(* CODESYS project rsCommTcpRt.library
   Company: ESO
   Description: This library provides generic drivers for Tcp Real-time communication.
      It also provides Local Control Device drivers for Tcp Real-time communication with Lakeshore 224 and 336.
      Depends on rsCommCommon.library
   Version: 0.2.0.3
   Placeholder: ESO LDC Comm Tcp RT Library
   Author: Dan Popovic
   Title: ESO LDC Comm Tcp RT Library

Project tree, tasks and I/O mapping:
  libraries: ESO LDC Comm Common Library, 0.2.0.3 (ESO); Tc2_Standard, * (Beckhoff Automation GmbH); Tc2_System, * (Beckhoff Automation GmbH); Tc2_Utilities, * (Beckhoff Automation GmbH); Tc3_Module, * (Beckhoff Automation GmbH); VisuDialogs, * (System); VisuSymbols, * (System)
  config/
    Lakeshore_RT_Ethernet_Adapter_InterfacePointer.jpg
    Lakeshore_RT_Ethernet_Adapter_Params.jpg
    Lakeshore_RT_Instance_OID_SymbolInitialization.png
  00000000-0000-0000-0000-000000000000|config\Lakeshore_RT_Ethernet_Adapter_InterfacePointer.jpg
  00000000-0000-0000-0000-000000000000|config\Lakeshore_RT_Ethernet_Adapter_Params.jpg
  00000000-0000-0000-0000-000000000000|config\Lakeshore_RT_Instance_OID_SymbolInitialization.png
  Data types/
    Enumerated/
      Comm/
        data type E_TCP_RT_CLIENT_STATUS
    Structures/
      Comm/
        data type T_TCP_RT_CLIENT_CFG
        data type T_TCP_RT_CLIENT_CTRL
        data type T_TCP_RT_CLIENT_INFO
        data type T_TCP_RT_CLIENT_STAT
        data type U_IpAdr
  Global Variables/
  lib/
  POUs/
    Comm/
      function block FB_TCP_RT_CLIENT [ST]: FB_exit, FB_init, FB_reinit, ReceiveData, ReceiveEvent, TcAddRef, TcQueryInterface, TcRelease
    Devices/
      function block FB_LAKESHORE_TCP_RT [ST]: ActivityInitializing, ActivityMonitoring, ActivityMonitoringUser, M_Configure, M_GetCouplerState, M_ReadFromReply, M_ReadSensors, M_UpdateStatus
    program MAIN [ST]
  Version/
    global variables Global_Version
  Visualizations/
    Templates/
      visualisation GUI_TEMPLATE_LAKESHORE_TCP_RT_224
      visualisation GUI_TEMPLATE_LAKESHORE_TCP_RT_336
    visualisation GUI_LAKESHORE_TCP_RT_224
    visualisation GUI_LAKESHORE_TCP_RT_336
  text list GlobalTextList
*)

// Data types/Enumerated/Comm/E_TCP_RT_CLIENT_STATUS
{attribute 'qualified_only'}
{attribute 'strict'}
TYPE E_TCP_RT_CLIENT_STATUS :
(
	NOT_INIT	:= -1,
	IDLE		:= 0,
	BUSY		:= 1,
	ERROR		:= 2
);
END_TYPE

// Data types/Structures/Comm/T_TCP_RT_CLIENT_CFG
TYPE T_TCP_RT_CLIENT_CFG :
STRUCT
	sTcpServerAdr:	STRING(16)	:= '62.159.14.51';	// Beckhoff Test-Website
    nTcpPort:    	UINT := 80;						// Beckhoff Test-Website
	

	// Parameters hidden from OPC UA access
	{attribute 'OPC.UA.DA' := '0'}
	tcpServerAdr:	U_IpAdr; 
END_STRUCT
END_TYPE

// Data types/Structures/Comm/T_TCP_RT_CLIENT_CTRL
TYPE T_TCP_RT_CLIENT_CTRL :
STRUCT
	bExecute: 	BOOL 	:= FALSE;
	sCmd:		STRING;
END_STRUCT
END_TYPE

// Data types/Structures/Comm/T_TCP_RT_CLIENT_INFO
TYPE T_TCP_RT_CLIENT_INFO :
STRUCT
(*
	Driver Information

	Change LOG:
	0.1.0.0		- First version.
*)

	sDate:			STRING(32)	:= '2018-10-09';
	sDescription:	STRING(80) 	:= 'TCP Client RT';
	sName:			STRING(64)	:= 'FB_TCP_CLIENT';
	sPlatform:		STRING(32)	:= 'CoDeSys';
	sSynopsis:		STRING(64)	:= 'TCP Client RT';
	nVersionMajor:	DINT		:= 0;
	nVersionMinor:	DINT		:= 1;

END_STRUCT
END_TYPE

// Data types/Structures/Comm/T_TCP_RT_CLIENT_STAT
TYPE T_TCP_RT_CLIENT_STAT :
STRUCT
	bInitialised:		BOOL	:= FALSE;		(* Flag if device is initialised *)


	nLastCommand:		DINT 	:= 0;
	nErrorCode:			DINT 	:= 0;
	nStatus: 			DINT	:= E_TCP_RT_CLIENT_STATUS.NOT_INIT;	// IDLE, BUSY, ERROR
	nCounter:			UDINT	:= 0;	// Alive counter

	sErrorText: 		STRING 	:= 'OK';
	sStatus:			STRING	:= '';	// Status description

	sLibVersion:		STRING	:= 'UNKNOWN';					(* Library version, e.g. '1.2.0.0' *)
	sSvnRevision:		STRING	:= '$$Revision: 311362 $$';		(* SVN Revision *)
	sRevision:			STRING	:= '';							(* SVN Revision without $ signs *)

	//Sample information about communication
    nReceivedPakets:	UINT;

	nSocketId:			UDINT; 
	nSentData:			UDINT; 

	bConnected:			BOOL	:= FALSE;
	nConnections: 		UDINT; 
	lastTcpEvent: 		TCPIP_EVENT;
	nReplyLength: 		UDINT; 
	sReply: 			STRING(255); 
	hrSend: 			HRESULT; //last SendData result

END_STRUCT
END_TYPE

// Data types/Structures/Comm/U_IpAdr
TYPE U_IpAdr :
UNION
	ipadrInternal : UDINT;
	ipadr : ARRAY[0..3] OF BYTE;
END_UNION
END_TYPE

// Version/Global_Version
{attribute 'TcGenerated'}
{attribute 'no-analysis'}
{attribute 'linkalways'}
// This function has been automatically generated from the project information.
VAR_GLOBAL CONSTANT
	{attribute 'const_non_replaced'}
	stLibVersion_ESO_LDC_Comm_Tcp_RT_Library : ST_LibVersion := (iMajor := 0, iMinor := 2, iBuild := 0, iRevision := 3, nFlags := 0, sVersion := '0.2.0.3');
END_VAR

// POUs/Comm/FB_TCP_RT_CLIENT
{attribute 'c++_compatible'}
FUNCTION_BLOCK FB_TCP_RT_CLIENT IMPLEMENTS ITcIoTcpProtocolRecv
VAR_INPUT
	{attribute 'OPC.UA.DA' := '0'}
	in_sDeviceTcpIpAdr:	STRING(16);	// Device IP address, e.g. '192.168.0.80'
	{attribute 'OPC.UA.DA' := '0'}
    in_nDeviceTcpPort:  UINT;		// Device Tcp port
END_VAR
VAR_OUTPUT
END_VAR
VAR
	{attribute 'OPC.UA.DA' := '1'}
	cfg:		T_TCP_RT_CLIENT_CFG;				// Config parameters
	{attribute 'OPC.UA.DA' := '1'}
	ctrl:		T_TCP_RT_CLIENT_CTRL;				// Control parameters
	{attribute 'OPC.UA.DA' := '1'}
	{attribute 'OPC.UA.DA.Access' := '1'}
	info:		T_TCP_RT_CLIENT_INFO; 				// Info parameters - ReadOnly
	{attribute 'OPC.UA.DA' := '1'}
	{attribute 'OPC.UA.DA.Access' := '1'}
	stat:		T_TCP_RT_CLIENT_STAT;				// Status parameters - ReadOnly


	// The following attribute has to be linked to corresponding Value 
	// of RT-Ethernet Adapter in Instance/'Symbol Initialization' tab
	{attribute 'TcInitSymbol'}
    oid: OTCID;	// Link to Value of RT-Ethernet Adapter in Instance/'Symbol Initialization' tab
	
    ipTcp:       ITcIoTcpProtocol;
	
	// Local variables
    ids: 	T_IPv4AddrArr;
	hrInit:	HRESULT; 
	
	// In case of error, try to allocate socket on every 100-th cycle.
	nSocketCounter:	UINT	:= 0;
	nSocketCounterLimit:	UINT	:= 100;
	

END_VAR

// TODO: Complete configuration
IF NOT stat.bInitialised THEN
	// Copy input parameters to config
	cfg.sTcpServerAdr	:= in_sDeviceTcpIpAdr;
	cfg.nTcpPort		:= in_nDeviceTcpPort;
	
	//generate Server IP adress
	ids := F_ScanIPv4AddrIds( in_sDeviceTcpIpAdr ); 
	cfg.tcpServerAdr.ipadr[3] := ids[0]; 
	cfg.tcpServerAdr.ipadr[2] := ids[1]; 
	cfg.tcpServerAdr.ipadr[1] := ids[2];
	cfg.tcpServerAdr.ipadr[0] := ids[3];
	
	// Get the version number 
	stat.sLibVersion	:= Global_Version.stLibVersion_ESO_LDC_Comm_Tcp_RT_Library.sVersion;
	stat.sRevision		:= MID(stat.sSvnRevision, LEN(stat.sSvnRevision)-2, 2);

	stat.bInitialised	:= TRUE;
	RETURN;
END_IF

IF(ipTcp <> 0) THEN 
	ipTcp.CheckReceived(); 
	IF (stat.nSocketId = 0) THEN 
		stat.bConnected	:= FALSE;
		nSocketCounter	:= nSocketCounter + 1;
		IF nSocketCounter > nSocketCounterLimit THEN
			nSocketCounter	:= 0;
			IF(ipTcp.AllocSocket(THIS^, stat.nSocketId) = 0) THEN //! THIS^ might get invalid due to online change! "Reallocate" by nSocketId <>0
				stat.nConnections := stat.nConnections+1;
				IF(ipTcp.Connect(stat.nSocketId, cfg.tcpServerAdr.ipadrInternal, cfg.nTcpPort) <> 0) THEN
					ipTcp.FreeSocket(stat.nSocketId); 
					stat.nSocketId := 0; 
				END_IF
			END_IF
		END_IF
	ELSE
		IF (ipTcp.IsConnected(stat.nSocketId) = S_OK) THEN 
			stat.bConnected	:= TRUE;
			IF ctrl.bExecute THEN
				ctrl.bExecute := FALSE;
				stat.hrSend := ipTcp.SendData(stat.nSocketId, INT_TO_UDINT(LEN(ctrl.sCmd)), ADR(ctrl.sCmd), stat.nSentData); 
			END_IF
		ELSE
			IF stat.bConnected THEN
				// We were connected but not any more.
				// Free the socket.
				ipTcp.FreeSocket(stat.nSocketId); 
				stat.nSocketId := 0; 
			END_IF
			stat.bConnected	:= FALSE;
		END_IF
	END_IF
END_IF

METHOD FB_exit : BOOL
VAR_INPUT
	bInCopyCode : BOOL; // if TRUE, the exit method is called for exiting an instance that is copied afterwards (online change).
END_VAR
IF NOT bInCopyCode THEN // no online change
	IF ipTcp <> 0 THEN 
		ipTcp.FreeSocket(stat.nSocketId); // Shutdown
		FW_SafeRelease(ADR(ipTcp));
		FB_exit := TRUE; 
	END_IF
END_IF
END_METHOD

METHOD FB_init : BOOL
VAR_INPUT
	bInitRetains: 	BOOL; // if TRUE, the retain variables are initialized (warm start / cold start)
	bInCopyCode: 	BOOL;  // if TRUE, the instance afterwards gets moved into the copy code (online change)
END_VAR
VAR
	ipSrv:	ITComObjectServer;
	
END_VAR
IF NOT bInCopyCode THEN // no online change
	IF ipTcp = 0 THEN
		hrInit := FW_ObjMgr_GetObjectInstance(	oid:=oid, 
												iid:=TC_GLOBAL_IID_LIST.IID_ITcIoTcpProtocol, 
												pipUnk:=ADR(ipTcp) );
		IF SUCCEEDED(hrInit) THEN
			FB_init := TRUE;
		ELSE 
			FW_SafeRelease(ADR(ipTcp));
		END_IF 
	END_IF
END_IF
END_METHOD

METHOD FB_reinit : BOOL
VAR_INPUT
END_VAR
IF (ipTcp <> 0 AND stat.nSocketId <> 0) THEN //reregister THIS^ for online changes  
	ipTcp.AllocSocket(THIS^, stat.nSocketId);
	FB_reinit := TRUE; 
END_IF
END_METHOD

{attribute 'object_name' := 'ReceiveData'}
{attribute 'c++_compatible'}
{attribute 'signature_flag' := '33554688'}
{attribute 'pack_mode' := '4'}
{attribute 'show'}
{attribute 'minimal_input_size' := '4'}
{attribute 'checksuperglobal'}
METHOD ReceiveData : HRESULT
VAR_INPUT
	socketId	: UDINT;
	nData	: UDINT;
	pData	: PVOID;
END_VAR
stat.nReceivedPakets	:= stat.nReceivedPakets+1;
stat.nReplyLength 		:= nData; //nonstripped

MEMCPY( ADR(stat.sReply), pData, MIN(nData, SIZEOF(stat.sReply)-1) );	//stripped to max length of string
memset(ADR(stat.sReply)+MIN(nData, SIZEOF(stat.sReply)-1)+1, 0, 1);		//add a 00 Byte at end of message
END_METHOD

{attribute 'object_name' := 'ReceiveEvent'}
{attribute 'c++_compatible'}
{attribute 'signature_flag' := '33554688'}
{attribute 'pack_mode' := '4'}
{attribute 'show'}
{attribute 'minimal_input_size' := '4'}
{attribute 'checksuperglobal'}
METHOD ReceiveEvent : HRESULT
VAR_INPUT
	socketId	: UDINT;
	tcpEvent	: TCPIP_EVENT;
END_VAR
stat.lastTcpEvent := tcpEvent;

CASE tcpEvent OF
	TCPIP_EVENT.TCPIP_EVENT_ERROR:
		stat.nStatus	:= E_TCP_RT_CLIENT_STATUS.ERROR;
		stat.sStatus	:= 'ERROR';
		ipTcp.FreeSocket(socketId);
		stat.nSocketId := 0; 
	TCPIP_EVENT.TCPIP_EVENT_RESET:
		stat.nStatus	:= E_TCP_RT_CLIENT_STATUS.BUSY;
		ipTcp.FreeSocket(socketId);
		stat.nSocketId := 0; 
	TCPIP_EVENT.TCPIP_EVENT_TIMEOUT:
		stat.nStatus	:= E_TCP_RT_CLIENT_STATUS.ERROR;
		stat.sStatus	:= 'TIMEOUT';
		ipTcp.FreeSocket(socketId);
		stat.nSocketId := 0; 
	TCPIP_EVENT.TCPIP_EVENT_CONN_CLOSED:
		ipTcp.FreeSocket(socketId);
		stat.nSocketId := 0; 
	TCPIP_EVENT.TCPIP_EVENT_CONN_INCOMING:
		stat.nStatus	:= E_TCP_RT_CLIENT_STATUS.BUSY;
	TCPIP_EVENT.TCPIP_EVENT_KEEP_ALIVE:
		stat.nStatus	:= E_TCP_RT_CLIENT_STATUS.BUSY;
	TCPIP_EVENT.TCPIP_EVENT_CONN_IDLE:
(*
		// Recovery
		IF ctrl.bExecute THEN
			ctrl.bExecute	:= FALSE;
			THIS^.ReceiveEvent(socketId,TCPIP_EVENT.TCPIP_EVENT_RESET);
		ELSE
			stat.nStatus	:= E_TCP_RT_CLIENT_STATUS.IDLE;
		END_IF
*)
	TCPIP_EVENT.TCPIP_EVENT_DATA_SENT:
		stat.sStatus	:= CONCAT(ctrl.sCmd, ' Sent');
	TCPIP_EVENT.TCPIP_EVENT_DATA_RECEIVED:
		stat.nStatus	:= E_TCP_RT_CLIENT_STATUS.IDLE;
		stat.sStatus	:= 'Data Received';
	(*
		IF nCmd = 1 THEN
			ctrl.sMessage	:= 'PID? 1$N';
			nCmd	:= 2;
		ELSIF nCmd = 2 THEN
			ctrl.sMessage	:= 'PID? 2$N';
			nCmd	:= 1;
		END_IF
		ctrl.bSend	:= TRUE;
		*)
//		THIS^.ReceiveEvent(socketId,TCPIP_EVENT.TCPIP_EVENT_CONN_IDLE);
	TCPIP_EVENT.TCPIP_EVENT_LINKCONNECT:
	// WARNING: Nothing to do?
	TCPIP_EVENT.TCPIP_EVENT_LINKDISCONNECT:
		ipTcp.FreeSocket(socketId);
		stat.nSocketId := 0; 
END_CASE; 
ReceiveEvent := S_OK;
END_METHOD

{attribute 'object_name' := 'TcAddRef'}
{attribute 'c++_compatible'}
{attribute 'signature_flag' := '33554688'}
{attribute 'pack_mode' := '4'}
{attribute 'show'}
{attribute 'minimal_input_size' := '4'}
{attribute 'checksuperglobal'}
METHOD TcAddRef : UDINT
END_METHOD

{attribute 'object_name' := 'TcQueryInterface'}
{attribute 'c++_compatible'}
{attribute 'signature_flag' := '33554688'}
{attribute 'pack_mode' := '4'}
{attribute 'show'}
{attribute 'minimal_input_size' := '4'}
{attribute 'checksuperglobal'}
METHOD TcQueryInterface : HRESULT
VAR_INPUT
	iid	: REFERENCE TO IID;
	pipItf	: POINTER TO PVOID;
END_VAR
VAR
	ipTcpRecv : ITcIoTcpProtocolRecv;
	ipUnknown : ITcUnknown;	
END_VAR
IF GuidsEqual(ADR(iid), ADR(TC_GLOBAL_IID_LIST.IID_ITcIoTcpProtocolRecv)) THEN
	ipTcpRecv := THIS^; // cast to interface pointer
	pipItf^ := ITCUNKNOWN_TO_PVOID(ipTcpRecv);
	TcAddRef();
	TcQueryInterface := S_OK;
ELSIF GuidsEqual(ADR(iid), ADR(TC_GLOBAL_IID_LIST.IID_ITcUnknown)) THEN
	ipUnknown := THIS^; // cast to interface pointer
	pipItf^ := ITCUNKNOWN_TO_PVOID(ipUnknown);
	TcAddRef();
	TcQueryInterface := S_OK;
ELSE
	TcQueryInterface := E_HRESULTAdsErr.NOINTERFACE ; //Call super if this fb extends some other
END_IF
END_METHOD

{attribute 'object_name' := 'TcRelease'}
{attribute 'c++_compatible'}
{attribute 'signature_flag' := '33554688'}
{attribute 'pack_mode' := '4'}
{attribute 'show'}
{attribute 'minimal_input_size' := '4'}
{attribute 'checksuperglobal'}
METHOD TcRelease : UDINT
END_METHOD

END_FUNCTION_BLOCK

// POUs/Devices/FB_LAKESHORE_TCP_RT
FUNCTION_BLOCK FB_LAKESHORE_TCP_RT EXTENDS FB_LAKESHORE_BASE
VAR_INPUT
	{attribute 'OPC.UA.DA' := '0'}
	in_sDeviceTcpIpAdr:	STRING(16);		// Lakeshore IP address, e.g. '192.168.0.80'
	{attribute 'OPC.UA.DA' := '0'}
    in_nDeviceTcpPort:  UINT := 7777;	// Lakeshore Tcp port, default 7777
END_VAR
VAR_OUTPUT
END_VAR
VAR CONSTANT
	// Monitoring states
	{attribute 'OPC.UA.DA' := '0'}
	C_STATE_SEND_CMD:			INT	:= 0;
	{attribute 'OPC.UA.DA' := '0'}
	C_STATE_DELAY_AFTER_SEND:	INT	:= 10;
	{attribute 'OPC.UA.DA' := '0'}
	C_STATE_WAIT_DATA_RECEIVED:	INT	:= 20;
	{attribute 'OPC.UA.DA' := '0'}
	C_STATE_WAIT:				INT	:= 30;
END_VAR
VAR

	{attribute 'OPC.UA.DA' := '0'}
	comm:		FB_TCP_RT_CLIENT;			// Instance of generic comm FB. OPC UA Disabled!!!

END_VAR


(* Execute comm instance *)
comm(	in_sDeviceTcpIpAdr:=in_sDeviceTcpIpAdr,
		in_nDeviceTcpPort:=in_nDeviceTcpPort);


// Execute the base class object FB_RS_BASE
SUPER^();

METHOD ActivityInitializing
VAR_INPUT
	bExecute:	BOOL;
END_VAR
VAR_INST
	{attribute 'OPC.UA.DA' := '0'}
    nMethodState:	INT := 0;	// State Machine current state
END_VAR
SetAction('ActivityInitializing');


IF NOT bExecute THEN
	nMethodState	:= 0;	// Reset the state machine
	cmdCounter		:= 1;	// Init will start from the first init command
	RETURN;
END_IF

// Handle State Machine
CASE nMethodState OF
	0:	// Set communication parameters and Model configuration
		(* Set comm suffixes for commands and replies *)
		// TODO: Suffix
//		ptrCommCfg^.sCmdSuffix		:= sCmdSuffix;
//		ptrCommCfg^.sReplySuffix	:= sReplySuffix;
		// Set Model and monitoring period (input parameters)
		cfg.nModel			:= in_nModel;
		cfg.bAutoMonitor	:= in_bAutoMonitor;
		cfg.tDelay_Periodic	:= DINT_TO_TIME(in_nPeriod);
		
		(* Pointers to INIT and READ commands set in M_Configure() depending on the model *)

		(* Set initial state and status *)
		stat.bInitialised	:= FALSE;
		stat.sReply			:= '';
		SetStatus(E_SM_ERROR.OK, 'BUSY');
		
		// DPO NEW START
		// Wait for connected
		fbTimer (IN := FALSE); (* Reset timer *)
		fbTimer (IN := TRUE, PT := T#10S); (* TODO: 80 sec timeout for reply *)
		nMethodState := 5;				// Go to next state, i.e. INIT_COMM
		RETURN;
		// DPO NEW END

		nMethodState := 10;				// Go to next state, i.e. INIT_COMM
		
		
	5:
		fbTimer (IN := TRUE);
		IF fbTimer.Q THEN
			// Timer expired after 5 sec. This is an error.
			fbTimer (IN := FALSE);
			SetStatus(E_LAKESHORE_ERROR.TIMEOUT, 'ERROR: Communication timeout');	
			bCommProblem	:= TRUE;
			nEvent := E_SM_EVENT.ERRINIT;
			RETURN;
		ELSIF comm.stat.bConnected THEN
			fbTimer (IN := FALSE);
			nMethodState := 10;				// Go to next state, i.e. INIT_COMM
		END_IF

	10:	// Initialize COMM port
		(* Reset the serial port *)
//		ptrCommCtrl^.nCommand	:= E_RS_COMM_CMD.INIT;
//		ptrCommCtrl^.bExecute	:= TRUE;

		(* Start the timer by going false/true *)
		fbTimer (IN := FALSE); (* Reset timer *)
		fbTimer (IN := TRUE, PT := T#20S); (* TODO: 80 sec timeout for reply *)

//		nMethodState 	:= 15;	// On next cycle wait until the comm port is reset, i.e. idle
		nMethodState 	:= 20;	// On next cycle wait until the comm port is reset, i.e. idle
		
	15:	// Wait for completion of command.
		// If command has no reply, wait for comm.stat.lastTcpEvent = TCPIP_EVENT.TCPIP_EVENT_DATA_SENT.
		// If it has, wait for               comm.stat.lastTcpEvent = TCPIP_EVENT.TCPIP_EVENT_DATA_RECEIVED.
		fbTimer (IN := TRUE);
		IF ((cfg.cmdList_Init[cmdCounter].nReplies = 0) AND 
			(comm.stat.lastTcpEvent = TCPIP_EVENT.TCPIP_EVENT_DATA_SENT OR 
			 comm.stat.lastTcpEvent = TCPIP_EVENT.TCPIP_EVENT_CONN_IDLE)) OR 
			((cfg.cmdList_Init[cmdCounter].nReplies > 0) AND 
			(comm.stat.lastTcpEvent = TCPIP_EVENT.TCPIP_EVENT_DATA_RECEIVED))THEN
			// Communication is IDLE 
			fbTimer (IN := FALSE);	// disable timer 
			stat.sReply		:= ptrCommStat^.sReply;	// Save the reply
			cmdCounter		:= cmdCounter + 1;	// Increment init command index
			fbTimer (IN := FALSE);	// disable timer 
			fbTimer (IN := TRUE, PT := cfg.tDelay_Init); // Wait INIT delay
			bCommProblem	:= FALSE;
			nMethodState 	:= 18;	// Execute next device INIT command
		ELSIF comm.stat.nStatus = E_RS_COMM_STATUS.ERROR THEN
			fbTimer (IN := FALSE);
			SetStatus(E_LAKESHORE_ERROR.COMM, 'ERROR: Communication error');	
			bCommProblem	:= TRUE;
			nEvent := E_SM_EVENT.ERRINIT;
			RETURN;
		ELSIF fbTimer.Q THEN
			// Timer expired after 5 sec. This is an error.
			fbTimer (IN := FALSE);
			SetStatus(E_LAKESHORE_ERROR.TIMEOUT, 'ERROR: Communication timeout');	
			bCommProblem	:= TRUE;
			nEvent := E_SM_EVENT.ERRINIT;
			RETURN;
		END_IF

	
	
	18:	// Wait INIT Delay
		fbTimer (IN := TRUE);
		IF fbTimer.Q THEN
			// Timer expired after 5 sec. This is an error.
			fbTimer (IN := FALSE);
			nMethodState 	:= 20;	// Execute next device INIT command
			RETURN;
		END_IF

	
	
	20:	// INIT DEV
		IF cfg.cmdList_Init[cmdCounter].cmd = '' THEN
			// Device INIT is done. Go to IDLE 
			stat.bInitialised 	:= TRUE;
			cmdCounter			:= 1;
			SetStatus(E_SM_ERROR.OK, 'IDLE');
			nEvent 		:= E_SM_EVENT.INITDONE;
			RETURN;
		END_IF
		
		(* Send INIT command with index cmdCounter *)
//		ptrCommCtrl^.nCommand		:= E_RS_COMM_CMD.SEND;
		ptrCommCtrl^.sCmd			:= CONCAT(cfg.cmdList_Init[cmdCounter].cmd,in_sCmdSuffix);
//		ptrCommCtrl^.nNumReplies	:= ptrInitCmds^ [cmdCounter].nReplies;
//		ptrCommCtrl^.bHasReply		:= ptrInitCmds^ [cmdCounter].nReplies > 0;
		ptrCommCtrl^.bExecute		:= TRUE;
	
		(* Start the timer by going false/true *)
		fbTimer (IN := FALSE); (* Reset timer *)
		fbTimer (IN := TRUE, PT := T#5S); (* 5 sec timeout for reply *)

		// On next cycle wait until the comm port is idle
		nMethodState 	:= 15;	// On next cycle wait until the comm port is idle
	
END_CASE
END_METHOD

METHOD ActivityMonitoring
VAR_INPUT
	bExecute:	BOOL;
END_VAR
VAR_INST
	{attribute 'OPC.UA.DA' := '0'}
    nMethodState:	INT := C_STATE_SEND_CMD;	// State Machine current state
	{attribute 'OPC.UA.DA' := '0'}
	nRetries:		INT := 0;	// Number of retries in case of communication problems
	{attribute 'OPC.UA.DA' := '0'}
	tDelay:			TIME	:= T#50MS;	// Min delay to wait after a command
END_VAR
IF NOT cfg.bAutoMonitor AND stat.nSubstate = E_RS_BASE_SUBSTATE.NOTOP_READY THEN
	SetAction('No Monitoring'); 
	SetStatus(E_SM_ERROR.OK, 'IDLE');
	nMethodState	:= C_STATE_SEND_CMD;	// Reset the state machine
	cmdCounter		:= 1;	// Reading will start from the first command in the array
	RETURN;
END_IF

IF NOT bExecute THEN
	SetAction('ActivityMonitoring'); 
//	SetStatus(E_SM_ERROR.OK, 'BUSY');
	nMethodState	:= C_STATE_SEND_CMD;	// Reset the state machine
	cmdCounter		:= 1;	// Reading will start from the first command in the array
	RETURN;
END_IF

// Handle State Machine
CASE nMethodState OF
	/////////////////
	C_STATE_SEND_CMD:	// Execute a command from the command array
	/////////////////
		IF cfg.cmdList_Read[cmdCounter].cmd = '' OR cmdCounter > 16 THEN
			// We arrived to the end of the array of pre-defined commands
			// Check if we have to exit Monitoring
			IF nReadType = E_RS_BASE_READ_TYPE.SINGLE	THEN
				// If it's a single read, exit here.
				SetStatus(E_SM_ERROR.OK, 'IDLE');
				nInternalEvent := E_SM_EVENT.READDONE;
				RETURN;
			END_IF

			// Periodic READ is done. Wait tDelay_Periodic before re-starting the READ.
			cmdCounter	:= 1;
			SetStatus(E_SM_ERROR.OK, 'IDLE');
			
			(* Start the timer by going false/true *)
			fbTimer (IN := FALSE); (* Reset timer *)
			fbTimer (IN := TRUE, PT := cfg.tDelay_Periodic);
			nMethodState := C_STATE_WAIT;				// Goto Wait for tDelay_Periodic
			RETURN;
		ELSIF NOT comm.stat.bConnected THEN
			SetStatus(E_LAKESHORE_ERROR.COMM, 'Send Failed.');	
			// Not connected yet. Don't do anything
			(* Start the timer by going false/true *)
			fbTimer (IN := FALSE); (* Reset timer *)
			fbTimer (IN := TRUE, PT := T#3S);
			nMethodState := C_STATE_WAIT;				// Goto Wait for tDelay_Periodic
			nEvent := E_SM_EVENT.ERRCOMM;
			RETURN;
		ELSE
			(* Send command with index cmdCounter *)
			ptrCommCtrl^.sCmd		:= CONCAT(cfg.cmdList_Read[cmdCounter].cmd,in_sCmdSuffix);
			ptrCommCtrl^.bExecute	:= TRUE;
			
			(* Start the timer by going false/true *)
			fbTimer (IN := FALSE); (* Reset timer *)
			fbTimer (IN := TRUE, PT := T#3MS); // 3 msec timeout before waiting for reply 
	
			nMethodState := C_STATE_DELAY_AFTER_SEND;	// Apply short WAIT for SEND to complete
		END_IF
		

		
	/////////////////////////
	C_STATE_DELAY_AFTER_SEND:	// Apply short WAIT for SEND to complete
	/////////////////////////
		fbTimer (IN := TRUE);

		(* If Timer has expired, go to the next state. *)
		IF fbTimer.Q THEN
			fbTimer (IN := FALSE);
			fbTimer (IN := TRUE, PT := T#5S); (* 5 sec timeout for reply *)
			SetStatus(E_SM_ERROR.OK, 'BUSY');
			nMethodState 	:= C_STATE_WAIT_DATA_RECEIVED;	// Goto Wait for TCPIP_EVENT_DATA_RECEIVED
			RETURN;
		END_IF
	

	///////////////////////////
	C_STATE_WAIT_DATA_RECEIVED:	// Wait for the reading to complete, i.e. TCPIP_EVENT_DATA_RECEIVED
	///////////////////////////
		fbTimer (IN := TRUE);
		IF	comm.stat.lastTcpEvent = TCPIP_EVENT.TCPIP_EVENT_DATA_RECEIVED THEN
			// Communication is IDLE 
			fbTimer (IN := FALSE);	// disable timer 
			stat.sReply		:= ptrCommStat^.sReply;	// Save the reply
			
			// Copy readings to status variable(s)
			
			// This was a single read.
			// The reply is already in stat.sReply.
			(* Store the last reading into stat.lrArrReadings array. The index is [cmdCounter] *)
			M_ReadFromReply(idx := DINT_TO_INT(cfg.cmdList_Read[cmdCounter].offset),
							n 	:= DINT_TO_INT(cfg.cmdList_Read[cmdCounter].nValues),
							str := stat.sReply,
							ok 	=> bResult);

			bCommProblem	:= FALSE;
			nRetries		:= 0;	// Reset number of retries

			
			cmdCounter		:= cmdCounter + 1;	// Reading will start from the first command in the array
			
			// Apply a short delay of 50 ms
			fbTimer (IN := FALSE); (* Reset timer *)
			fbTimer (IN := TRUE, PT := tDelay);
			nMethodState := C_STATE_WAIT;	// Goto WAIT for IDLE
			nEvent := E_SM_EVENT.COMMOK;
			RETURN;
		ELSIF NOT comm.stat.bConnected OR comm.stat.nStatus = E_RS_COMM_STATUS.ERROR OR fbTimer.Q THEN
			// There is a communication problem.
			// Try to recover by waiting for 5 sec and retrying.
			fbTimer (IN := FALSE);
			bCommProblem	:= TRUE;
			// Increase Retry count
			nRetries		:= nRetries + 1;		// Increment number of retries
			stat.nRetries	:= stat.nRetries + 1;	// Increment total number of retries
			SetStatus(E_LAKESHORE_ERROR.COMM, 'Receive failed');	
			nEvent := E_SM_EVENT.ERRCOMM;	
			cmdCounter	:= 1;	// Start from the first command
			// Apply a long delay of 1 sec and then retry.
			fbTimer (IN := FALSE); (* Reset timer *)
			fbTimer (IN := TRUE, PT := T#1S);
			nMethodState	:= C_STATE_WAIT;	// wait a bit
			RETURN;
		END_IF


	//////////////////
	C_STATE_WAIT:	// Wait until the timer expires
	//////////////////
		fbTimer (IN := TRUE);

		// Check if we have to exit Monitoring
		IF nNextState <> E_RS_BASE_STATE.NONE THEN
			fbTimer (IN := FALSE); (* Stop the timer *)
			SetStatus(E_SM_ERROR.OK, nNextDescription);
			SetState(nNextState, nNextSubstate);
			nNextState		:= E_RS_BASE_STATE.NONE;
			nNextSubstate	:= E_RS_BASE_SUBSTATE.NONE;
			nNextDescription:= '';
			RETURN;
		END_IF
	
		(* If Timer has expired, go to the next state. *)
		IF fbTimer.Q	THEN
			fbTimer (IN := FALSE);
//			SetStatus(E_SM_ERROR.OK, 'BUSY');
			statRef.sErrorText 	:= 'BUSY';
			nMethodState 	:= C_STATE_SEND_CMD;	// Goto SEND command
			RETURN;
		END_IF
	

	
END_CASE
END_METHOD

METHOD ActivityMonitoringUser
VAR_INPUT
	bExecute:	BOOL;
END_VAR
VAR_INST
	{attribute 'OPC.UA.DA' := '0'}
    nMethodState:	INT := 0;	// State Machine current state
	{attribute 'OPC.UA.DA' := '0'}
	nRetries:		INT := 0;	// Number of retries in case of communication problems
END_VAR

IF NOT bExecute THEN
	SetAction('ActivityMonitoringUser'); 
	SetStatus(E_SM_ERROR.OK, 'BUSY');
	nMethodState	:= 0;	// Reset the state machine
	RETURN;
END_IF

// Handle State Machine
CASE nMethodState OF
	0:	// Execute the User command ctrl.sCmdUser.cmd
		
//		ptrCommCtrl^.nCommand		:= E_RS_COMM_CMD.SEND;
		ptrCommCtrl^.sCmd			:= ctrl.sCmdUser.cmd;
//		ptrCommCtrl^.nNumReplies	:= ctrl.sCmdUser.nReplies;
//		ptrCommCtrl^.bHasReply		:= ctrl.sCmdUser.nReplies > 0;
		ptrCommCtrl^.bExecute		:= TRUE;
		
		(* Start the timer by going false/true *)
		fbTimer (IN := FALSE); (* Reset timer *)
		fbTimer (IN := TRUE, PT := T#5S); (* 5 sec timeout for reply *)

		nMethodState := 20;				// Goto WAIT for Reading to complete,

	10:	// Wait until the delay timeout expires
		fbTimer (IN := TRUE);

		// Check if we have to exit Monitoring
		IF nNextState <> E_RS_BASE_STATE.NONE THEN
			fbTimer (IN := FALSE); (* Stop the timer *)
			SetStatus(E_SM_ERROR.OK, nNextDescription);
			SetState(nNextState, nNextSubstate);
			nNextState		:= E_RS_BASE_STATE.NONE;
			nNextSubstate	:= E_RS_BASE_SUBSTATE.NONE;
			nNextDescription:= '';
			RETURN;
		END_IF
	
		(* If Timer has expired, go to the next state. *)
		IF fbTimer.Q THEN
			fbTimer (IN := FALSE);
			SetStatus(E_SM_ERROR.OK, 'BUSY');
			nMethodState 	:= 0;				// Goto Wait for tDelay_Periodic
			RETURN;
		END_IF
	


	20:	// Wait for the reading to complete, i.e. IDLE
		fbTimer (IN := TRUE);
		IF comm.stat.nStatus = E_RS_COMM_STATUS.IDLE THEN
			// Communication is IDLE 
			fbTimer (IN := FALSE);	// disable timer 
			
			// Save the reply. That's all since we don't know how too process the reply
			stat.sReplyUser	:= ptrCommStat^.sReply;	
			
			bCommProblem	:= FALSE;
			nRetries		:= 0;	// Reset number of retries

			
			// Check if we have to exit Monitoring
			IF nNextState <> E_RS_BASE_STATE.NONE THEN
				fbTimer (IN := FALSE); (* Stop the timer *)
				SetStatus(E_SM_ERROR.OK, nNextDescription);
				SetState(nNextState, nNextSubstate);
				nNextState		:= E_RS_BASE_STATE.NONE;
				nNextSubstate	:= E_RS_BASE_SUBSTATE.NONE;
				nNextDescription:= '';
				RETURN;
			ELSIF nReadType <> E_RS_BASE_READ_TYPE.PERIODIC_USER	THEN
				// This was single READ_USER
				SetStatus(E_SM_ERROR.OK, 'IDLE');
				nInternalEvent := E_SM_EVENT.READDONE;
				RETURN;
			ELSE
				// Periodic READ is done. Wait tDelay_Periodic before re-starting the READ.
				SetStatus(E_SM_ERROR.OK, 'IDLE');
				
				(* Start the timer by going false/true *)
				fbTimer (IN := FALSE); (* Reset timer *)
				fbTimer (IN := TRUE, PT := cfg.tDelay_Periodic);
				nMethodState := 10;				// Goto Wait for tDelay_Periodic
			END_IF
			RETURN;
		ELSIF comm.stat.nStatus = E_RS_COMM_STATUS.ERROR OR fbTimer.Q THEN
			fbTimer (IN := FALSE);
			SetStatus(E_LAKESHORE_ERROR.COMM, 'ERROR: Communication error');	
			bCommProblem	:= TRUE;
			// Retry up to 3 times
			nRetries		:= nRetries + 1;		// Increment number of retries
			stat.nRetries	:= stat.nRetries + 1;	// Increment total number of retries
			IF nRetries > 3 THEN
				nEvent := E_SM_EVENT.ERRCOMM;
			ELSE
				// Apply a short delay of 1 sec and retry
				fbTimer (IN := FALSE); (* Reset timer *)
				fbTimer (IN := TRUE, PT := T#1000MS);
				nMethodState := 10;				// Goto Wait 
			END_IF
			RETURN;
		END_IF

	
END_CASE
END_METHOD

METHOD M_Configure
VAR_INPUT
END_VAR
VAR
	// This is OK for models 224 and 336
	cmdList_Init_224:	ARRAY [1..8] OF T_LAKESHORE_COMMAND := [
							(cmd := 'MODE 1', 	nReplies := 0, 	nValues := 0,	offset := 0),
							(cmd := '*IDN?', 	nReplies := 1, 	nValues := 1,	offset := 0),
							(cmd := '', 		nReplies := 0, 	nValues := 0,	offset := 0),
							(cmd := '', 		nReplies := 0, 	nValues := 0,	offset := 0),
							(cmd := '', 		nReplies := 0, 	nValues := 0,	offset := 0),
							(cmd := '', 		nReplies := 0, 	nValues := 0,	offset := 0),
							(cmd := '', 		nReplies := 0, 	nValues := 0,	offset := 0),
							(cmd := '', 		nReplies := 0, 	nValues := 0,	offset := 0)];

	cmdList_Init_336:	ARRAY [1..8] OF T_LAKESHORE_COMMAND := [
							(cmd := 'MODE 1', 	nReplies := 0, 	nValues := 0,	offset := 0),
							(cmd := '*IDN?', 	nReplies := 1, 	nValues := 1,	offset := 0),
							(cmd := '', 		nReplies := 0, 	nValues := 0,	offset := 0),
							(cmd := '', 		nReplies := 0, 	nValues := 0,	offset := 0),
							(cmd := '', 		nReplies := 0, 	nValues := 0,	offset := 0),
							(cmd := '', 		nReplies := 0, 	nValues := 0,	offset := 0),
							(cmd := '', 		nReplies := 0, 	nValues := 0,	offset := 0),
							(cmd := '', 		nReplies := 0, 	nValues := 0,	offset := 0)];


	(*	List of READ commands *)
	(* Lakeshore 218 commands:
		Command "KRDG? 0" requests all 8 temperature values in K.
		Command "CRDG? 0" requests all 8 temperature values in C.
		Reply format: 
			+nn.nnn,+nn.nnn,+nn.nnn,+nn.nnn,+nn.nnn,+nn.nnn,+nn.nnn,+nn.nnn<CR><LF>
	*)

	cmdList_Read_224:	ARRAY [1..16] OF T_LAKESHORE_COMMAND := [
							(cmd := 'KRDG? 0', 	nReplies := 1, 	nValues := 12,	offset := 0),
							(cmd := 'CRDG? 0', 	nReplies := 1, 	nValues := 12,	offset := 12),
							(cmd := '', 		nReplies := 0, 	nValues := 0,	offset := 0),
							(cmd := '', 		nReplies := 0, 	nValues := 0,	offset := 0),
							(cmd := '', 		nReplies := 0, 	nValues := 0,	offset := 0),
							(cmd := '', 		nReplies := 0, 	nValues := 0,	offset := 0),
							(cmd := '', 		nReplies := 0, 	nValues := 0,	offset := 0),
							(cmd := '', 		nReplies := 0, 	nValues := 0,	offset := 0),
							(cmd := '', 		nReplies := 0, 	nValues := 0,	offset := 0),
							(cmd := '', 		nReplies := 0, 	nValues := 0,	offset := 0),
							(cmd := '', 		nReplies := 0, 	nValues := 0,	offset := 0),
							(cmd := '', 		nReplies := 0, 	nValues := 0,	offset := 0),
							(cmd := '', 		nReplies := 0, 	nValues := 0,	offset := 0),
							(cmd := '', 		nReplies := 0, 	nValues := 0,	offset := 0),
							(cmd := '', 		nReplies := 0, 	nValues := 0,	offset := 0),
							(cmd := '', 		nReplies := 0, 	nValues := 0,	offset := 0)];

	cmdList_Read_336:	ARRAY [1..16] OF T_LAKESHORE_COMMAND := [
							(cmd := 'KRDG? A', 	nReplies := 1, 	nValues := 1,	offset := 0),
							(cmd := 'KRDG? B', 	nReplies := 1, 	nValues := 1,	offset := 1),
							(cmd := 'SETP? 1', 	nReplies := 1, 	nValues := 1,	offset := 2),
							(cmd := 'PID? 1', 	nReplies := 1, 	nValues := 3,	offset := 3),
							(cmd := 'RAMP? 1', 	nReplies := 1, 	nValues := 2,	offset := 6),
							(cmd := 'RANGE? 1', nReplies := 1, 	nValues := 1,	offset := 8),
							(cmd := 'HTR? 1', 	nReplies := 1, 	nValues := 1,	offset := 9),
							(cmd := 'SETP? 2', 	nReplies := 1, 	nValues := 1,	offset := 10),
							(cmd := 'PID? 2', 	nReplies := 1, 	nValues := 3,	offset := 11),
							(cmd := 'RAMP? 2', 	nReplies := 1, 	nValues := 2,	offset := 14),
							(cmd := 'RANGE? 2', nReplies := 1, 	nValues := 1,	offset := 16),
							(cmd := 'HTR? 2', 	nReplies := 1, 	nValues := 1,	offset := 17),
							(cmd := 'AOUT? 3', 	nReplies := 1, 	nValues := 1,	offset := 18),
							(cmd := 'AOUT? 4', 	nReplies := 1, 	nValues := 1,	offset := 19),
							(cmd := '', 		nReplies := 0, 	nValues := 0,	offset := 0),
							(cmd := '', 		nReplies := 0, 	nValues := 0,	offset := 0)];

	
END_VAR
// Execute base FB M_Configure().
// This will set cfg.nModel
SUPER^.M_Configure();

// TODO
// Populate cfg.cmdList_Init and cmdList_Read tables for the specific cfg.nModel.
IF cfg.nModel = 224 THEN
	cfg.cmdList_Init	:= cmdList_Init_224;
	cfg.cmdList_Read	:= cmdList_Read_224;
ELSIF cfg.nModel = 336 THEN
	cfg.cmdList_Init	:= cmdList_Init_336;
	cfg.cmdList_Read	:= cmdList_Read_336;
END_IF


// Set pointers to comm, i.e.
ptrCommCfg	:= ADR(comm.cfg);	(* Pointer to comm.cfg instance *)
ptrCommCtrl	:= ADR(comm.ctrl);	(* Pointer to comm.ctrl instance *)
ptrCommStat	:= ADR(comm.stat);	(* Pointer to comm.stat instance *)

// Set comm suffixes for commands and replies
ptrCommCfg^.sCmdSuffix		:= in_sCmdSuffix;
ptrCommCfg^.sReplySuffix	:= in_sReplySuffix;
END_METHOD

METHOD M_GetCouplerState : BOOL
VAR_INPUT
END_VAR
M_GetCouplerState	:= TRUE;
END_METHOD

METHOD M_ReadFromReply : BOOL
(* FB to extract 'n' values from 'str' and copy them into stat.lrArrReadings starting from index 'idx'.

	Example: 
		M_ReadFromReply (	idx := 5, 
							n := 3, 
							str := '0050.1,0020.2,0000$0D$0A', 
							ok => ok);
		res [5] = 50.1
		res [6] = 20.2
		res [7] = 0.0
		ok = TRUE
*)

VAR_INPUT
	idx:	INT;		(* arr [idx] will hold the first extracted value, arr [idx+1] the second one, etc. *)
	n:		INT;		(* Number of values to extract from the string - command specific *)
	str:	STRING(255);		(* String returned in Lakeshore reply *)
END_VAR
VAR_OUTPUT
	ok:		BOOL;		(* TRUE if the reading was correct, i.e. 'n' values successfully extracted from 'str'.  *)
END_VAR

VAR
	i:		INT;
	str_l:	STRING(255);
	pos:	INT;
END_VAR
i	:= 0;
str_l	:= str;
ok	:= TRUE; (* OK *)


WHILE i < n DO
	stat.lrArrReadings [idx + i].lrValue	:= STRING_TO_LREAL (str_l); (* take the first number *)
	(* move to just after the comma *)
	IF i < (n-1) THEN
		pos := FIND (str_l, ','); (* find the comma *)
		IF pos = 0 THEN (* less than 'n' numbers present in the string *)
			ok	:= FALSE; (* ERROR *)
			i 	:= n;
		ELSE
			str_l := RIGHT (str_l, LEN(str_l) - pos);
			i	:= i + 1;
		END_IF
	ELSE
		i	:= i + 1;
	END_IF
END_WHILE
END_METHOD

METHOD M_ReadSensors
VAR_INPUT
END_VAR
VAR
	i:	int;
END_VAR
//
// Digital inputs are mapped to physical input signals.
// Assign preconfigured label depending on the value
//
//FOR i := 0 TO (cfg.nNumInDig - 1) DO
//	arrDI[i].M_Compute();
//END_FOR
END_METHOD

METHOD M_UpdateStatus
VAR_INPUT
END_VAR
// TODO
//
// Copy values from stat.lrReadings to correspondig stat variables.
// Check M_Configure(). It has to match!
//
// This is an example for model 340.
// This method has to match the list of commands in T_LAKESHORE_CFG::cmdList_Read
IF cfg.nModel = 224 THEN
	// Nothing to do.
	// NOTE: 12 readings [K]: stat.lrArrReadings[0..11].lrValue
	// NOTE: 12 readings [C]: stat.lrArrReadings[12..23].lrValue
	;	
ELSIF cfg.nModel = 336 THEN
	// TODO NOTE: Only loop 1 is handled !!!
	stat.lrKRDG_A		:= stat.lrArrReadings[0].lrValue;
	stat.lrCRDG_A		:= stat.lrKRDG_A - 273.15;
	stat.lrKRDG_B		:= stat.lrArrReadings[1].lrValue;
	stat.lrCRDG_B		:= stat.lrKRDG_B - 273.15;
	// Loop 1
	stat.lrSETP			:= stat.lrArrReadings[2].lrValue;
	stat.nPID_P			:= LREAL_TO_UINT(stat.lrArrReadings[3].lrValue);
	stat.nPID_I			:= LREAL_TO_UINT(stat.lrArrReadings[4].lrValue);
	stat.nPID_D			:= LREAL_TO_UINT(stat.lrArrReadings[5].lrValue);
	stat.bRAMP_On		:= LREAL_TO_BOOL(stat.lrArrReadings[6].lrValue);
	stat.lrRAMP_Rate	:= stat.lrArrReadings[7].lrValue;
	stat.nRANGE			:= LREAL_TO_UINT(stat.lrArrReadings[8].lrValue);
	stat.lrHTR			:= stat.lrArrReadings[9].lrValue;
	// Loop 2
	stat.lrSETP2		:= stat.lrArrReadings[10].lrValue;
	stat.nPID2_P		:= LREAL_TO_UINT(stat.lrArrReadings[11].lrValue);
	stat.nPID2_I		:= LREAL_TO_UINT(stat.lrArrReadings[12].lrValue);
	stat.nPID2_D		:= LREAL_TO_UINT(stat.lrArrReadings[13].lrValue);
	stat.bRAMP2_On		:= LREAL_TO_BOOL(stat.lrArrReadings[14].lrValue);
	stat.lrRAMP2_Rate	:= stat.lrArrReadings[15].lrValue;
	stat.nRANGE			:= LREAL_TO_UINT(stat.lrArrReadings[16].lrValue);
	stat.lrHTR			:= stat.lrArrReadings[17].lrValue;
	// Outputs
	stat.lrAOUT3		:= stat.lrArrReadings[18].lrValue;
	stat.lrAOUT4		:= stat.lrArrReadings[19].lrValue;

END_IF
END_METHOD

END_FUNCTION_BLOCK

// POUs/MAIN
PROGRAM MAIN
VAR
	// Lakeshore 224 (Ethernet TCP Realtime interface)
	{attribute 'OPC.UA.DA' := '1'}
	LS224_TCP_RT:	FB_LAKESHORE_TCP_RT;	// LakeShore based on FB_TCP_RT_CLIENT

	// Lakeshore 336 (Ethernet TCP Realtime interface)
	{attribute 'OPC.UA.DA' := '1'}
	LS336_TCP_RT:	FB_LAKESHORE_TCP_RT;	// LakeShore based on FB_TCP_RT_CLIENT
	
	bDymmy	AT %I*:	BOOL;

END_VAR

		
LS224_TCP_RT(	in_sName			:= 'LS224_TCP_RT',
				in_nModel			:= 224,
				in_sCmdSuffix		:= '$0D$0A',
				in_sDeviceTcpIpAdr	:= '192.168.0.12',
				in_nDeviceTcpPort	:= 7777,
				in_nPeriod			:= 1200); 
		
LS336_TCP_RT(	in_sName			:= 'LS336_TCP_RT',
				in_nModel			:= 336,
				in_sCmdSuffix		:= '$0A',
				in_sDeviceTcpIpAdr	:= '192.168.0.80',
				in_nDeviceTcpPort	:= 7777,
				in_nPeriod			:= 1000);

END_PROGRAM

// Visualizations/Templates/GUI_TEMPLATE_LAKESHORE_TCP_RT_224
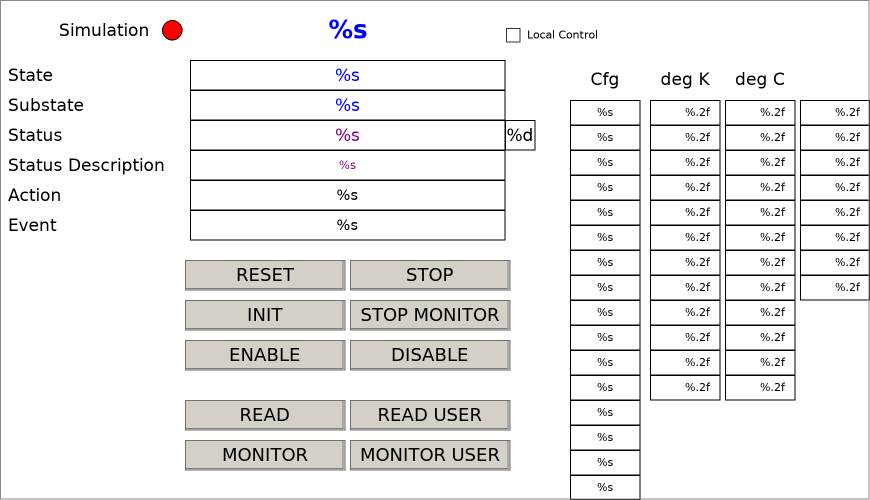
VISUALIZATION GUI_TEMPLATE_LAKESHORE_TCP_RT_224  // 870x500
VAR_IN_OUT
	m_Instance:	FB_LAKESHORE_TCP_RT;
END_VAR
    Rectangle (190,60 315x30), "%s", text variable: m_Instance.stat.sState
    Rectangle (190,90 315x30), "%s", text variable: m_Instance.stat.sSubstate
    Button (185,260 160x30), "RESET", input disabled if: (m_Instance.stat.bLocal = FALSE) <> 0
        OnMouseClick: execute { m_Instance.ctrl.nCommand := E_RS_COMMAND.RESET; m_Instance.ctrl.bExecute := TRUE; }
    Button (185,300 160x30), "INIT", input disabled if: (m_Instance.stat.bLocal = FALSE) <> 0
        OnMouseClick: execute { m_Instance.ctrl.nCommand := E_RS_COMMAND.INIT; m_Instance.ctrl.bExecute := TRUE; }
    Button (350,260 160x30), "STOP", input disabled if: (m_Instance.stat.bLocal = FALSE) <> 0
        OnMouseClick: execute { m_Instance.ctrl.nCommand := E_RS_COMMAND.STOP; m_Instance.ctrl.bExecute := TRUE; }
    Button (185,340 160x30), "ENABLE", input disabled if: (m_Instance.stat.bLocal = FALSE) <> 0
        OnMouseClick: execute { m_Instance.ctrl.nCommand := E_RS_COMMAND.ENABLE; m_Instance.ctrl.bExecute := TRUE; }
    Button (350,340 160x30), "DISABLE", input disabled if: (m_Instance.stat.bLocal = FALSE) <> 0
        OnMouseClick: execute { m_Instance.ctrl.nCommand := E_RS_COMMAND.DISABLE; m_Instance.ctrl.bExecute := TRUE; }
    Rectangle (5,60 180x30), "State"
    Rectangle (5,90 180x30), "Substate"
    Rectangle (190,120 315x30), "%s", text variable: m_Instance.stat.sStatus
    Rectangle (190,150 315x30), "%s", text variable: m_Instance.stat.sErrorText
    Rectangle (5,120 180x30), "Status"
    Rectangle (5,150 180x30), "Status Description"
    Rectangle (190,180 315x30), "%s", text variable: m_Instance.stat.sActionDesc
    Rectangle (190,210 315x30), "%s", text variable: m_Instance.stat.sEventDesc
    Rectangle (5,180 180x30), "Action"
    Rectangle (5,210 180x30), "Event"
    Rectangle (232,12 232x35), "%s", text variable: m_Instance.in_sName
    Rectangle (574,64 62x30), "Cfg"
    Checkbox (504,20 116x30), "Local Control", variable: m_Instance.stat.bLocal
    Rectangle (505,120 30x30), "%d", text variable: m_Instance.stat.nStatus
    Button (185,400 160x30), "READ", tooltip "Single read of all commands in the configuration", input disabled if: (m_Instance.stat.bLocal = FALSE) <> 0
        OnMouseClick: execute { m_Instance.ctrl.nCommand := E_RS_COMMAND.READ; m_Instance.ctrl.bExecute := TRUE; }
    Button (350,400 160x30), "READ USER", tooltip "Single read of user command", input disabled if: (m_Instance.stat.bLocal = FALSE) <> 0
        OnMouseClick: execute { m_Instance.ctrl.nCommand := E_RS_COMMAND.READ_USER; m_Instance.ctrl.bExecute := TRUE; }
    Button (185,440 160x30), "MONITOR", tooltip "Continuously read all commands in the configuration", input disabled if: (m_Instance.stat.bLocal = FALSE) <> 0
        OnMouseClick: execute { m_Instance.ctrl.nCommand := E_RS_COMMAND.MONITOR; m_Instance.ctrl.bExecute := TRUE; }
    Button (350,440 160x30), "MONITOR USER", tooltip "Continuously read the User command", input disabled if: (m_Instance.stat.bLocal = FALSE) <> 0
        OnMouseClick: execute { m_Instance.ctrl.nCommand := E_RS_COMMAND.MONITOR_USER; m_Instance.ctrl.bExecute := TRUE; }
    Rectangle (570,100 70x25), "%s", text variable: m_Instance.cfg.cmdList_Read[1].cmd
    Rectangle (570,125 70x25), "%s", text variable: m_Instance.cfg.cmdList_Read[2].cmd
    Rectangle (570,150 70x25), "%s", text variable: m_Instance.cfg.cmdList_Read[3].cmd
    Rectangle (570,175 70x25), "%s", text variable: m_Instance.cfg.cmdList_Read[4].cmd
    Rectangle (570,200 70x25), "%s", text variable: m_Instance.cfg.cmdList_Read[5].cmd
    Rectangle (570,225 70x25), "%s", text variable: m_Instance.cfg.cmdList_Read[6].cmd
    Rectangle (570,250 70x25), "%s", text variable: m_Instance.cfg.cmdList_Read[7].cmd
    Rectangle (570,275 70x25), "%s", text variable: m_Instance.cfg.cmdList_Read[8].cmd
    Rectangle (570,300 70x25), "%s", text variable: m_Instance.cfg.cmdList_Read[9].cmd
    Rectangle (570,325 70x25), "%s", text variable: m_Instance.cfg.cmdList_Read[10].cmd
    Rectangle (570,350 70x25), "%s", text variable: m_Instance.cfg.cmdList_Read[11].cmd
    Rectangle (570,375 70x25), "%s", text variable: m_Instance.cfg.cmdList_Read[12].cmd
    Rectangle (570,400 70x25), "%s", text variable: m_Instance.cfg.cmdList_Read[13].cmd
    Rectangle (570,425 70x25), "%s", text variable: m_Instance.cfg.cmdList_Read[14].cmd
    Rectangle (570,450 70x25), "%s", text variable: m_Instance.cfg.cmdList_Read[15].cmd
    Rectangle (570,475 70x25), "%s", text variable: m_Instance.cfg.cmdList_Read[16].cmd
    Rectangle (650,100 70x25), "%.2f", text variable: m_Instance.stat.lrArrReadings[0].lrValue
    Rectangle (650,125 70x25), "%.2f", text variable: m_Instance.stat.lrArrReadings[1].lrValue
    Rectangle (650,150 70x25), "%.2f", text variable: m_Instance.stat.lrArrReadings[2].lrValue
    Rectangle (650,175 70x25), "%.2f", text variable: m_Instance.stat.lrArrReadings[3].lrValue
    Rectangle (650,200 70x25), "%.2f", text variable: m_Instance.stat.lrArrReadings[4].lrValue
    Rectangle (650,225 70x25), "%.2f", text variable: m_Instance.stat.lrArrReadings[5].lrValue
    Rectangle (650,250 70x25), "%.2f", text variable: m_Instance.stat.lrArrReadings[6].lrValue
    Rectangle (650,275 70x25), "%.2f", text variable: m_Instance.stat.lrArrReadings[7].lrValue
    Rectangle (650,350 70x25), "%.2f", text variable: m_Instance.stat.lrArrReadings[8].lrValue
    Rectangle (650,375 70x25), "%.2f", text variable: m_Instance.stat.lrArrReadings[9].lrValue
    Rectangle (650,300 70x25), "%.2f", text variable: m_Instance.stat.lrArrReadings[10].lrValue
    Rectangle (650,325 70x25), "%.2f", text variable: m_Instance.stat.lrArrReadings[11].lrValue
    Rectangle (725,100 70x25), "%.2f", text variable: m_Instance.stat.lrArrReadings[12].lrValue
    Rectangle (725,125 70x25), "%.2f", text variable: m_Instance.stat.lrArrReadings[13].lrValue
    Rectangle (725,150 70x25), "%.2f", text variable: m_Instance.stat.lrArrReadings[14].lrValue
    Rectangle (725,175 70x25), "%.2f", text variable: m_Instance.stat.lrArrReadings[15].lrValue
    Rectangle (725,200 70x25), "%.2f", text variable: m_Instance.stat.lrArrReadings[16].lrValue
    Rectangle (725,225 70x25), "%.2f", text variable: m_Instance.stat.lrArrReadings[17].lrValue
    Rectangle (725,250 70x25), "%.2f", text variable: m_Instance.stat.lrArrReadings[18].lrValue
    Rectangle (725,275 70x25), "%.2f", text variable: m_Instance.stat.lrArrReadings[19].lrValue
    Rectangle (654,64 62x30), "deg K"
    Rectangle (729,64 62x30), "deg C"
    Rectangle (725,300 70x25), "%.2f", text variable: m_Instance.stat.lrArrReadings[20].lrValue
    Rectangle (725,325 70x25), "%.2f", text variable: m_Instance.stat.lrArrReadings[21].lrValue
    Rectangle (725,350 70x25), "%.2f", text variable: m_Instance.stat.lrArrReadings[22].lrValue
    Rectangle (725,375 70x25), "%.2f", text variable: m_Instance.stat.lrArrReadings[23].lrValue
    Rectangle (800,100 70x25), "%.2f", text variable: m_Instance.stat.lrArrReadings[24].lrValue
    Rectangle (800,125 70x25), "%.2f", text variable: m_Instance.stat.lrArrReadings[25].lrValue
    Rectangle (800,150 70x25), "%.2f", text variable: m_Instance.stat.lrArrReadings[26].lrValue
    Rectangle (800,175 70x25), "%.2f", text variable: m_Instance.stat.lrArrReadings[27].lrValue
    Rectangle (800,200 70x25), "%.2f", text variable: m_Instance.stat.lrArrReadings[28].lrValue
    Rectangle (800,225 70x25), "%.2f", text variable: m_Instance.stat.lrArrReadings[29].lrValue
    Rectangle (800,250 70x25), "%.2f", text variable: m_Instance.stat.lrArrReadings[30].lrValue
    Rectangle (800,275 70x25), "%.2f", text variable: m_Instance.stat.lrArrReadings[31].lrValue
    Button (350,300 160x30), "STOP MONITOR", tooltip "Stop Monitoring if in OP/MONITORIN state.", input disabled if: (m_Instance.stat.bLocal = FALSE) <> 0
        OnMouseClick: execute { m_Instance.ctrl.nCommand := E_RS_COMMAND.STOPMON; m_Instance.ctrl.bExecute := TRUE; }
    Rectangle (56,15 101x30), "Simulation", invisible if: (m_Instance.stat.bSimulation=FALSE)
    Ellipse (162,20 20x20), tooltip "GREEN=Initialized RED=Not-initialized", text variable: m_Instance.stat.bInitialised, invisible if: (m_Instance.stat.bSimulation=FALSE)
END_VISUALIZATION

// Visualizations/Templates/GUI_TEMPLATE_LAKESHORE_TCP_RT_336
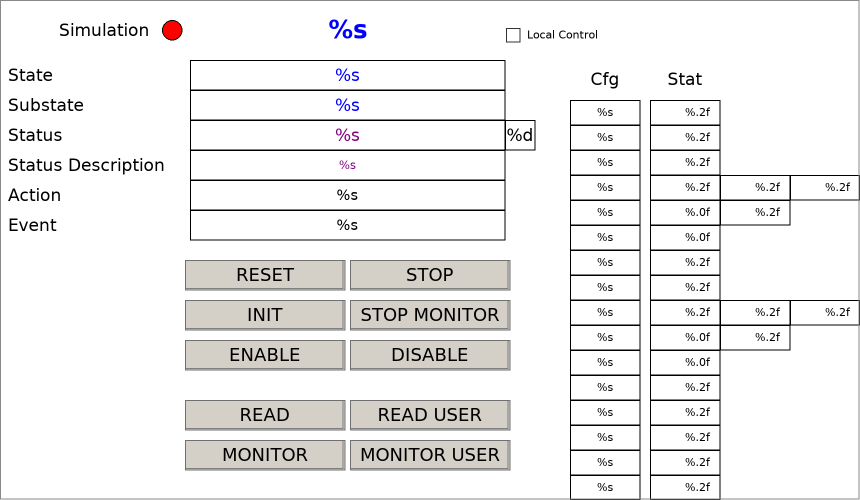
VISUALIZATION GUI_TEMPLATE_LAKESHORE_TCP_RT_336  // 860x500
VAR_IN_OUT
	m_Instance:	FB_LAKESHORE_TCP_RT;
END_VAR
    Rectangle (190,60 315x30), "%s", text variable: m_Instance.stat.sState
    Rectangle (190,90 315x30), "%s", text variable: m_Instance.stat.sSubstate
    Button (185,260 160x30), "RESET", input disabled if: (m_Instance.stat.bLocal = FALSE) <> 0
        OnMouseClick: execute { m_Instance.ctrl.nCommand := E_RS_COMMAND.RESET; m_Instance.ctrl.bExecute := TRUE; }
    Button (185,300 160x30), "INIT", input disabled if: (m_Instance.stat.bLocal = FALSE) <> 0
        OnMouseClick: execute { m_Instance.ctrl.nCommand := E_RS_COMMAND.INIT; m_Instance.ctrl.bExecute := TRUE; }
    Button (350,260 160x30), "STOP", input disabled if: (m_Instance.stat.bLocal = FALSE) <> 0
        OnMouseClick: execute { m_Instance.ctrl.nCommand := E_RS_COMMAND.STOP; m_Instance.ctrl.bExecute := TRUE; }
    Button (185,340 160x30), "ENABLE", input disabled if: (m_Instance.stat.bLocal = FALSE) <> 0
        OnMouseClick: execute { m_Instance.ctrl.nCommand := E_RS_COMMAND.ENABLE; m_Instance.ctrl.bExecute := TRUE; }
    Button (350,340 160x30), "DISABLE", input disabled if: (m_Instance.stat.bLocal = FALSE) <> 0
        OnMouseClick: execute { m_Instance.ctrl.nCommand := E_RS_COMMAND.DISABLE; m_Instance.ctrl.bExecute := TRUE; }
    Rectangle (5,60 180x30), "State"
    Rectangle (5,90 180x30), "Substate"
    Rectangle (190,120 315x30), "%s", text variable: m_Instance.stat.sStatus
    Rectangle (190,150 315x30), "%s", text variable: m_Instance.stat.sErrorText
    Rectangle (5,120 180x30), "Status"
    Rectangle (5,150 180x30), "Status Description"
    Rectangle (190,180 315x30), "%s", text variable: m_Instance.stat.sActionDesc
    Rectangle (190,210 315x30), "%s", text variable: m_Instance.stat.sEventDesc
    Rectangle (5,180 180x30), "Action"
    Rectangle (5,210 180x30), "Event"
    Rectangle (232,12 232x35), "%s", text variable: m_Instance.in_sName
    Rectangle (574,64 62x30), "Cfg"
    Checkbox (504,20 116x30), "Local Control", variable: m_Instance.stat.bLocal
    Rectangle (505,120 30x30), "%d", text variable: m_Instance.stat.nStatus
    Button (185,400 160x30), "READ", tooltip "Single read of all commands in the configuration", input disabled if: (m_Instance.stat.bLocal = FALSE) <> 0
        OnMouseClick: execute { m_Instance.ctrl.nCommand := E_RS_COMMAND.READ; m_Instance.ctrl.bExecute := TRUE; }
    Button (350,400 160x30), "READ USER", tooltip "Single read of user command", input disabled if: (m_Instance.stat.bLocal = FALSE) <> 0
        OnMouseClick: execute { m_Instance.ctrl.nCommand := E_RS_COMMAND.READ_USER; m_Instance.ctrl.bExecute := TRUE; }
    Button (185,440 160x30), "MONITOR", tooltip "Continuously read all commands in the configuration", input disabled if: (m_Instance.stat.bLocal = FALSE) <> 0
        OnMouseClick: execute { m_Instance.ctrl.nCommand := E_RS_COMMAND.MONITOR; m_Instance.ctrl.bExecute := TRUE; }
    Button (350,440 160x30), "MONITOR USER", tooltip "Continuously read the User command", input disabled if: (m_Instance.stat.bLocal = FALSE) <> 0
        OnMouseClick: execute { m_Instance.ctrl.nCommand := E_RS_COMMAND.MONITOR_USER; m_Instance.ctrl.bExecute := TRUE; }
    Rectangle (570,100 70x25), "%s", text variable: m_Instance.cfg.cmdList_Read[1].cmd
    Rectangle (570,125 70x25), "%s", text variable: m_Instance.cfg.cmdList_Read[2].cmd
    Rectangle (570,150 70x25), "%s", text variable: m_Instance.cfg.cmdList_Read[3].cmd
    Rectangle (570,175 70x25), "%s", text variable: m_Instance.cfg.cmdList_Read[4].cmd
    Rectangle (570,200 70x25), "%s", text variable: m_Instance.cfg.cmdList_Read[5].cmd
    Rectangle (570,225 70x25), "%s", text variable: m_Instance.cfg.cmdList_Read[6].cmd
    Rectangle (570,250 70x25), "%s", text variable: m_Instance.cfg.cmdList_Read[7].cmd
    Rectangle (570,275 70x25), "%s", text variable: m_Instance.cfg.cmdList_Read[8].cmd
    Rectangle (570,300 70x25), "%s", text variable: m_Instance.cfg.cmdList_Read[9].cmd
    Rectangle (570,325 70x25), "%s", text variable: m_Instance.cfg.cmdList_Read[10].cmd
    Rectangle (570,350 70x25), "%s", text variable: m_Instance.cfg.cmdList_Read[11].cmd
    Rectangle (570,375 70x25), "%s", text variable: m_Instance.cfg.cmdList_Read[12].cmd
    Rectangle (570,400 70x25), "%s", text variable: m_Instance.cfg.cmdList_Read[13].cmd
    Rectangle (570,425 70x25), "%s", text variable: m_Instance.cfg.cmdList_Read[14].cmd
    Rectangle (570,450 70x25), "%s", text variable: m_Instance.cfg.cmdList_Read[15].cmd
    Rectangle (570,475 70x25), "%s", text variable: m_Instance.cfg.cmdList_Read[16].cmd
    Rectangle (650,100 70x25), "%.2f", text variable: m_Instance.stat.lrArrReadings[0].lrValue
    Rectangle (650,125 70x25), "%.2f", text variable: m_Instance.stat.lrArrReadings[1].lrValue
    Rectangle (650,150 70x25), "%.2f", text variable: m_Instance.stat.lrArrReadings[2].lrValue
    Rectangle (650,175 70x25), "%.2f", text variable: m_Instance.stat.lrArrReadings[3].lrValue
    Rectangle (720,175 70x25), "%.2f", text variable: m_Instance.stat.lrArrReadings[4].lrValue
    Rectangle (790,175 70x25), "%.2f", text variable: m_Instance.stat.lrArrReadings[5].lrValue
    Rectangle (650,200 70x25), "%.0f", text variable: m_Instance.stat.lrArrReadings[6].lrValue
    Rectangle (650,225 70x25), "%.0f", text variable: m_Instance.stat.lrArrReadings[8].lrValue
    Rectangle (650,250 70x25), "%.2f", text variable: m_Instance.stat.lrArrReadings[9].lrValue
    Rectangle (650,275 70x25), "%.2f", text variable: m_Instance.stat.lrArrReadings[10].lrValue
    Rectangle (720,300 70x25), "%.2f", text variable: m_Instance.stat.lrArrReadings[12].lrValue
    Rectangle (790,300 70x25), "%.2f", text variable: m_Instance.stat.lrArrReadings[13].lrValue
    Rectangle (650,300 70x25), "%.2f", text variable: m_Instance.stat.lrArrReadings[11].lrValue
    Rectangle (720,325 70x25), "%.2f", text variable: m_Instance.stat.lrArrReadings[15].lrValue
    Rectangle (650,350 70x25), "%.0f", text variable: m_Instance.stat.lrArrReadings[16].lrValue
    Rectangle (650,375 70x25), "%.2f", text variable: m_Instance.stat.lrArrReadings[17].lrValue
    Rectangle (650,400 70x25), "%.2f", text variable: m_Instance.stat.lrArrReadings[18].lrValue
    Rectangle (650,425 70x25), "%.2f", text variable: m_Instance.stat.lrArrReadings[19].lrValue
    Rectangle (650,450 70x25), "%.2f", text variable: m_Instance.stat.lrArrReadings[20].lrValue
    Rectangle (650,475 70x25), "%.2f", text variable: m_Instance.stat.lrArrReadings[21].lrValue
    Rectangle (654,64 62x30), "Stat"
    Button (350,300 160x30), "STOP MONITOR", tooltip "Stop Monitoring if in OP/MONITORIN state.", input disabled if: (m_Instance.stat.bLocal = FALSE) <> 0
        OnMouseClick: execute { m_Instance.ctrl.nCommand := E_RS_COMMAND.STOPMON; m_Instance.ctrl.bExecute := TRUE; }
    Rectangle (56,15 101x30), "Simulation", invisible if: (m_Instance.stat.bSimulation=FALSE)
    Ellipse (162,20 20x20), tooltip "GREEN=Initialized RED=Not-initialized", text variable: m_Instance.stat.bInitialised, invisible if: (m_Instance.stat.bSimulation=FALSE)
    Rectangle (720,200 70x25), "%.2f", text variable: m_Instance.stat.lrArrReadings[7].lrValue
    Rectangle (650,325 70x25), "%.0f", text variable: m_Instance.stat.lrArrReadings[14].lrValue
END_VISUALIZATION

// Visualizations/GUI_LAKESHORE_TCP_RT_224
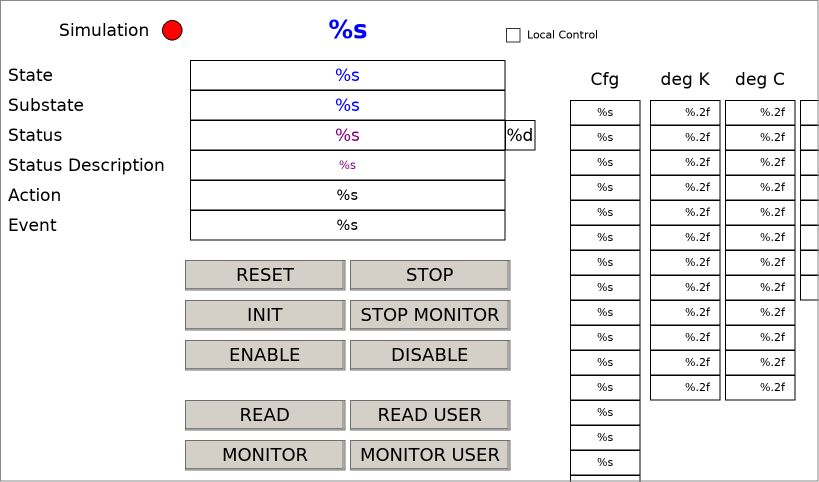
VISUALIZATION GUI_LAKESHORE_TCP_RT_224  // 819x482
    Frame (0,0 817x480)
        shows GUI_TEMPLATE_LAKESHORE_TCP_RT_224(m_Instance := MAIN.LS224_TCP_RT)
END_VISUALIZATION

// Visualizations/GUI_LAKESHORE_TCP_RT_336
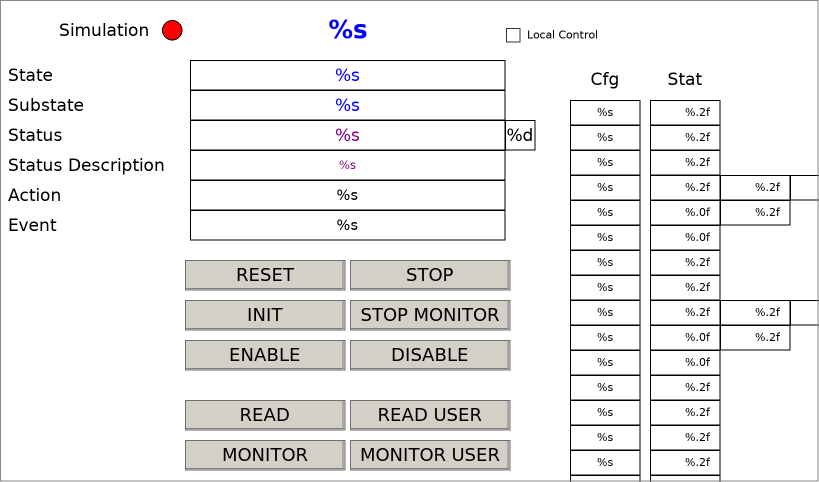
VISUALIZATION GUI_LAKESHORE_TCP_RT_336  // 819x482
    Frame (0,0 817x480)
        shows GUI_TEMPLATE_LAKESHORE_TCP_RT_336(m_Instance := MAIN.LS336_TCP_RT)
END_VISUALIZATION
